(* Logix 5000 project; controller Drives_Line1 1756-L72 rev 20.13; software revision 20.04; part 6 of 21 *)
(* tags used below, declared in another part *)
   EntryCtrl : UDT_Control_Zone;
   In_Commands : UDT_Commands;
   In_Config : UDT_Config;
   In_Setpoints : UDT_Setpoints;
   LineCmd : UDT_Commands_Line;
   Out_Feedbacks : UDT_Fdbks;
   Out_Status : UDT_Status;
   TestConfig_Unwinder_1 : UDT_Config_Unwinder;
   Unwinder_1 : UDT_Unwinder;
   Unwinder_2 : UDT_Unwinder;
   zConfigFromMaster : BOOL;
(* P10_Unwinder_1, continued *)

ROUTINE R98_ToDrive   (* ladder *)
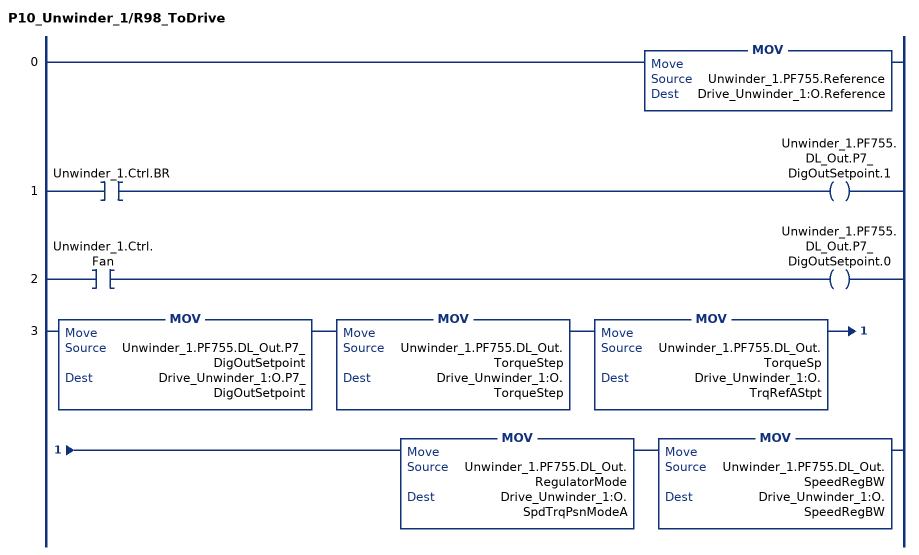
   0: MOV(Unwinder_1.PF755.Reference,Drive_Unwinder_1:O.Reference);
   1: XIC(Unwinder_1.Ctrl.BR)OTE(Unwinder_1.PF755.DL_Out.P7_DigOutSetpoint.1);
   2: XIC(Unwinder_1.Ctrl.Fan)OTE(Unwinder_1.PF755.DL_Out.P7_DigOutSetpoint.0);
   3: MOV(Unwinder_1.PF755.DL_Out.P7_DigOutSetpoint,Drive_Unwinder_1:O.P7_DigOutSetpoint)MOV(Unwinder_1.PF755.DL_Out.TorqueStep,Drive_Unwinder_1:O.TorqueStep)MOV(Unwinder_1.PF755.DL_Out.TorqueSp,Drive_Unwinder_1:O.TrqRefAStpt)MOV(Unwinder_1.PF755.DL_Out.RegulatorMode,Drive_Unwinder_1:O.SpdTrqPsnModeA)MOV(Unwinder_1.PF755.DL_Out.SpeedRegBW,Drive_Unwinder_1:O.SpeedRegBW);
END_ROUTINE

ROUTINE R999_Test   (* ladder *)
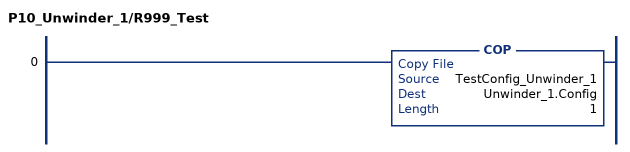
   0: COP(TestConfig_Unwinder_1,Unwinder_1.Config,1);
END_ROUTINE

ROUTINE R99_To_Master   (* ladder *)
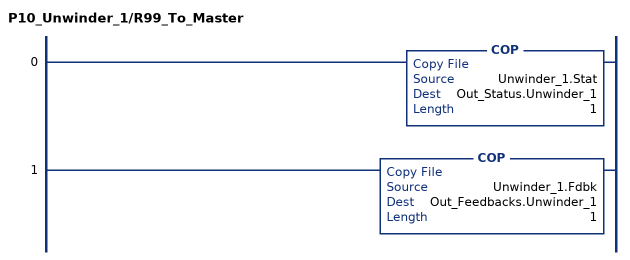
   0: COP(Unwinder_1.Stat,Out_Status.Unwinder_1,1);
   1: COP(Unwinder_1.Fdbk,Out_Feedbacks.Unwinder_1,1);
END_ROUTINE
END_PROGRAM

PROGRAM P11_Unwinder_2   (* main routine R00_Main *)
VAR
   ABS_01 : FBD_MATH_ADVANCED; {access Read Only}
   ABS_02 : FBD_MATH_ADVANCED;
   ABS_03 : FBD_MATH_ADVANCED;
   ABS_04 : FBD_MATH_ADVANCED;
   ADD_03 : FBD_MATH;
   BAND_01 : FBD_BOOLEAN_AND := (In3 := 1, In4 := 1, In5 := 1, In6 := 1, In7 := 1, In8 := 1);
   BAND_02 : FBD_BOOLEAN_AND := (In4 := 1, In5 := 1, In6 := 1, In7 := 1, In8 := 1);
   BAND_03 : FBD_BOOLEAN_AND := (In3 := 1, In4 := 1, In5 := 1, In6 := 1, In7 := 1, In8 := 1);
   BAND_04 : FBD_BOOLEAN_AND := (In3 := 1, In4 := 1, In5 := 1, In6 := 1, In7 := 1, In8 := 1);
   BAND_05 : FBD_BOOLEAN_AND := (In3 := 1, In4 := 1, In5 := 1, In6 := 1, In7 := 1, In8 := 1);
   BAND_06 : FBD_BOOLEAN_AND := (In1 := 1, In3 := 1, In4 := 1, In5 := 1, In6 := 1, In7 := 1, In8 := 1);
   BAND_07 : FBD_BOOLEAN_AND := (In3 := 1, In4 := 1, In5 := 1, In6 := 1, In7 := 1, In8 := 1);
   BAND_08 : FBD_BOOLEAN_AND := (In3 := 1, In4 := 1, In5 := 1, In6 := 1, In7 := 1, In8 := 1);
   BAND_09 : FBD_BOOLEAN_AND := (In3 := 1, In4 := 1, In5 := 1, In6 := 1, In7 := 1, In8 := 1);
   BNOT_01 : FBD_BOOLEAN_NOT := (Out := 1);
   BNOT_02 : FBD_BOOLEAN_NOT := (Out := 1);
   BNOT_04 : FBD_BOOLEAN_NOT := (Out := 1);
   BNOT_06 : FBD_BOOLEAN_NOT := (Out := 1);
   BNOT_07 : FBD_BOOLEAN_NOT := (Out := 1);
   BNOT_08 : FBD_BOOLEAN_NOT := (Out := 1);
   BOR_01 : FBD_BOOLEAN_OR := (In1 := 1, Out := 1);
   BOR_02 : FBD_BOOLEAN_OR;
   BOR_03 : FBD_BOOLEAN_OR;
   Diamtest : BOOL;
   Diamtest_mm : REAL := 725.0;
   DIV_01 : FBD_MATH := (SourceA := 2.5, SourceB := 100.0, Dest := 0.025);
   DIV_02 : FBD_MATH := (SourceB := 78.0);
   DIV_04 : FBD_MATH := (SourceB := 1440.0);
   DIV_10 : FBD_MATH := (Dest := 1770.7737);
   DIV_11 : FBD_MATH := (SourceA := 1770.7737, SourceB := 3.1415927, Dest := 563.6547);
   DIV_12 : FBD_MATH := (SourceB := 60.0);
   DIV_14 : FBD_MATH := (SourceB := 0.00494885);
   DIV_15 : FBD_MATH := (SourceA := 50.0, SourceB := 100.0, Dest := 0.5);
   EQU_01 : FBD_COMPARE := (SourceA := 1.0, SourceB := 4.0);
   FGEN_01 : FUNCTION_GENERATOR := (XY1Size := 21);
   GEQ_02 : FBD_COMPARE := (SourceB := 0.5);
   GRT_01 : FBD_COMPARE := (SourceB := 1.e-04);
   HLL_01 : HL_LIMIT := (In := 563.14075, HighLimit := 2000.0, LowLimit := 500.0, Out := 563.14075);
   HLL_07 : HL_LIMIT := (In := 6500.0, HighLimit := 15000.0, LowLimit := 1.0, Out := 6500.0);
   INTG_01 : INTEGRATOR := (Initialize := 1, IGain := 1000.02, RTSTime := 1, DeltaT := 0.05);
   INTG_02 : INTEGRATOR := (Initialize := 1, IGain := 0.016666, RTSTime := 1, DeltaT := 0.05);
   IO_State_Tmp_Unwinder_2 : INT := 16384;
   IO_State_Unwinder_2 : INT := 4;
   LES_01 : FBD_COMPARE;
   LPF_02 : FILTER_LOW_PASS := (WLag := 10.0, Order := 1, RTSTime := 1, DeltaT := 0.05); {access Read Only}
   LPF_1000 : FILTER_LOW_PASS := (WLag := 10.0, Order := 1, RTSTime := 1, DeltaT := 0.05);
   LPF_1006 : FILTER_LOW_PASS := (WLag := 10.0, Order := 1, RTSTime := 1, DeltaT := 0.05);
   MUL_01 : FBD_MATH := (SourceB := 2645.3247);
   MUL_02 : FBD_MATH := (SourceB := 0.00494885);
   MUL_03 : FBD_MATH := (SourceB := 25.0);
   MUL_04 : FBD_MATH := (SourceB := 100.0);
   MUL_05 : FBD_MATH := (SourceB := 0.5);
   MUL_06 : FBD_MATH := (SourceA := 5.0, SourceB := 0.5, Dest := 2.5);
   MUL_07 : FBD_MATH := (SourceA := 1.0065495);
   MUL_23 : FBD_MATH := (SourceA := 6500.0, SourceB := 0.5, Dest := 3250.0);
   MUL_26 : FBD_MATH := (SourceB := 2645.3247);
   NEG_01 : FBD_MATH_ADVANCED := (Source := 0.083, Dest := -0.083);
   NEG_03 : FBD_MATH_ADVANCED;
   NEG_04 : FBD_MATH_ADVANCED;
   NEG_06 : FBD_MATH_ADVANCED;
   RLIM_01 : RATE_LIMITER := (In := 563.6547, RTSTime := 1, Out := 563.14075, DeltaT := 0.05);
   RLIM_03 : RATE_LIMITER := (IncRate := 0.25, DecRate := 0.25, RTSTime := 1, DeltaT := 0.05);
   RLIM_04 : RATE_LIMITER := (IncRate := 5000.0, DecRate := 5000.0, ByPass := 1, RTSTime := 1, DeltaT := 0.05);
   SCL_01 : SCALE := (In := 562.0898, InRawMax := 5851.2163, InEUMax := 35.0, InEUMin := 25.0, Limiting := 1, Out := 25.960638);
   SCL_02 : SCALE := (InRawMax := 0.5, InEUMax := 10.0, InEUMin := 5.0, Limiting := 1, Out := 5.0);
   SCRV_02 : S_CURVE := (Initialize := 1, AbsAlgRamp := 1, AccelRate := 0.16, DecelRate := 0.16, JerkRate := 0.25, RTSTime := 1, DeltaT := 0.05);
   SEL_02 : SELECT := (In2 := 0.025);
   SEL_03 : SELECT;
   SEL_04 : SELECT;
   SEL_05 : SELECT := (In1 := 563.6547, In2 := 800.0, Out := 563.6547);
   SEL_06 : SELECT := (In1 := 563.14075, In2 := 725.0, Out := 563.14075);
   SEL_07 : SELECT := (In1 := 0.5, In2 := 0.5, Out := 0.5);
   SEL_08 : SELECT := (In1 := 563.6547, In2 := 800.0, Out := 563.6547);
   SEL_10 : SELECT;
   SEL_18 : SELECT := (In1 := 6500.0, SelectorIn := 1);
   SSUM_01 : SELECTED_SUMMER := (In1 := 0.083, Gain1 := 1.0, In2 := -0.083, Gain2 := 1.0, Gain3 := 1.0, Select3 := 1, Gain4 := 1.0, Gain5 := 1.0, Gain6 := 1.0, Gain7 := 1.0, Gain8 := 1.0);
   SSUM_02 : SELECTED_SUMMER := (Gain1 := 1.0, Select1 := 1, Gain2 := 1.0, Gain3 := 1.0, Gain4 := 1.0, Gain5 := 1.0, Gain6 := 1.0, Gain7 := 1.0, Gain8 := 1.0);
   SSUM_03 : SELECTED_SUMMER := (Gain1 := 1.0, Select1 := 1, Gain2 := 1.0, Gain3 := 1.0, Gain4 := 1.0, Gain5 := 1.0, Gain6 := 1.0, Gain7 := 1.0, Gain8 := 1.0);
   SSUM_05 : SELECTED_SUMMER := (Gain1 := 1.0, Gain2 := 1.0, Gain3 := 1.0, Gain4 := 1.0, Gain5 := 1.0, Gain6 := 1.0, Gain7 := 1.0, Gain8 := 1.0);
   SUB_08 : FBD_MATH; {access Read Only}
   TimeForBr : TIMER := (PRE := 750);
   TimeOffBr : TIMER := (PRE := 2000, ACC := 2000);
   TimeOffFan : TIMER := (PRE := 180000, ACC := 180000);
   TofReset : TIMER := (PRE := 1000, ACC := 1000);
   TonLowTension : TIMER := (PRE := 2500);
   TonNoResponse : TIMER := (PRE := 2500);
   TonRefOn : TIMER := (PRE := 500);
   TonTensionOnSp : TIMER := (PRE := 500);
   Unwind_1_DiamCalcOn : BOOL;
   Unwinder_2_JEC : REAL := 1.0; {access Read Only}
   Unwinder_2_JLossCrvSpd : REAL[21] := ([0] := -1500.0, [1] := -1350.0, [2] := -1200.0, [3] := -1050.0, [4] := -900.0, [5] := -750.0, [6] := -600.0, [7] := -450.0, [8] := -300.0, [9] := -150.0, [11] := 150.0, [12] := 300.0, [13] := 450.0, [14] := 600.0, [15] := 750.0, [16] := 900.0, [17] := 1050.0, [18] := 1200.0, [19] := 1350.0, [20] := 1500.0);
   Unwinder_2_JMaterial : REAL := 0.006549485; {access Read Only}
   Unwinder_2_LossCrvTrq_Pct : REAL[21] := ([0] := -6.0, [1] := -6.7, [2] := -6.7, [3] := -6.7, [4] := -6.7, [5] := -6.7, [6] := -6.5, [7] := -6.0, [8] := -5.0, [9] := -1.5, [11] := 2.0, [12] := 6.0, [13] := 6.8, [14] := 7.5, [15] := 7.5, [16] := 7.5, [17] := 7.5, [18] := 7.5, [19] := 7.5, [20] := 6.5);
   Unwinder_2_MatMass : REAL := 562.0898; {access Read Only}
   Unwinder_2_MatVolume : REAL := 0.15089658; {access Read Only}
   Unwinder_2_MaxMass : REAL := 5851.2163;
   Unwinder_2_MaxVolume : REAL := 1.5707964;
   Unwinder_2_PctPerN : REAL := 0.00494885; {access Read Only}
   Unwinder_2_RatedTrq : REAL := 72.94375; {access Read Only}
   Unwinder_2_RPMPerMPS : REAL := 2645.3247;
   Unwinder_2_SpdMps_Flt : REAL;
   Unwinder_2_SpdRpm_Flt : REAL;
   zUnwind_2_MaxRate : REAL := 0.25;
   zUnwind_2_TenRefRate : REAL := 5000.0;
   zUnwind_2_TenSpStall : REAL := 50.0;
   zUnwind_2_TrqTrimLimMax_Pct : REAL := 10.0;
   zUnwind_2_TrqTrimLimMin_Pct : REAL := 5.0;
   zUnwinder_2_JGainQ1Q2 : REAL := 0.5;
   zUnwinder_2_JGainQ3Q4 : REAL := 0.5;
   zUnwinder_2_SpdReg_BWMax : REAL := 35.0;
   zUnwinder_2_SpdReg_BWmin : REAL := 25.0;
   zUnwinder_2_Stall_Spd : REAL := 5.0;
   zUnwinder_2_Tens_Offs : REAL := 100.0;
END_VAR

ROUTINE R00_Main   (* ladder *)
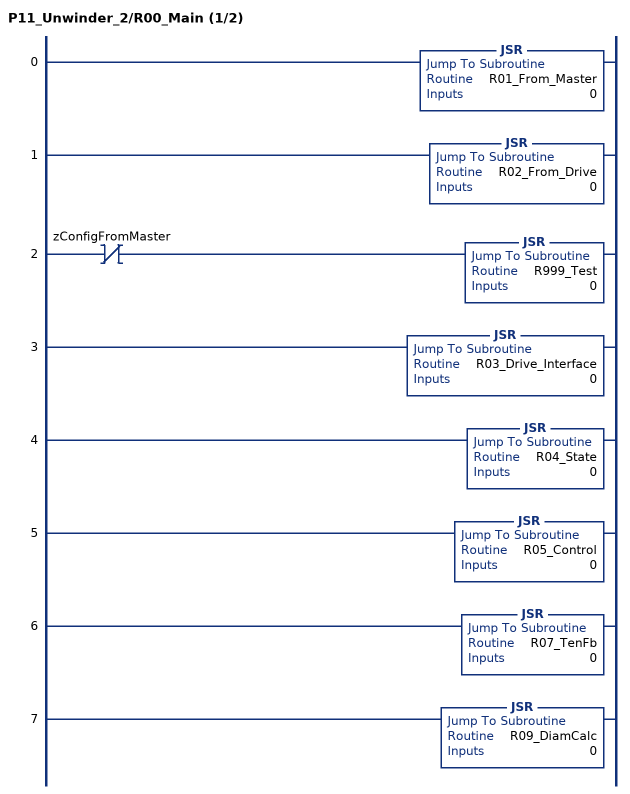
   0: JSR(R01_From_Master,0);
   1: JSR(R02_From_Drive,0);
   2: XIO(zConfigFromMaster)JSR(R999_Test,0);
   3: JSR(R03_Drive_Interface,0);
   4: JSR(R04_State,0);
   5: JSR(R05_Control,0);
   6: JSR(R07_TenFb,0);
   7: JSR(R09_DiamCalc,0);
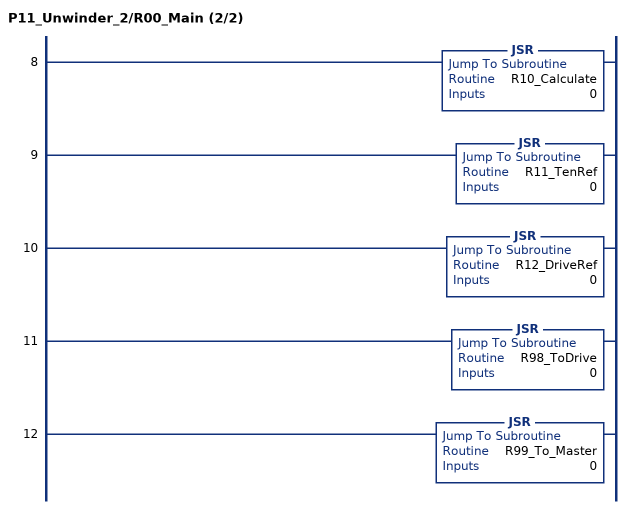
   8: JSR(R10_Calculate,0);
   9: JSR(R11_TenRef,0);
   10: JSR(R12_DriveRef,0);
   11: JSR(R98_ToDrive,0);
   12: JSR(R99_To_Master,0);
END_ROUTINE

ROUTINE R01_From_Master   (* ladder *)
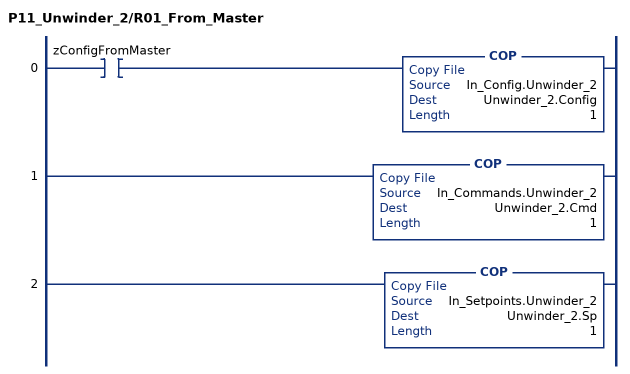
   0: XIC(zConfigFromMaster)COP(In_Config.Unwinder_2,Unwinder_2.Config,1);
   1: COP(In_Commands.Unwinder_2,Unwinder_2.Cmd,1);
   2: COP(In_Setpoints.Unwinder_2,Unwinder_2.Sp,1);
END_ROUTINE

ROUTINE R02_From_Drive   (* ladder *)
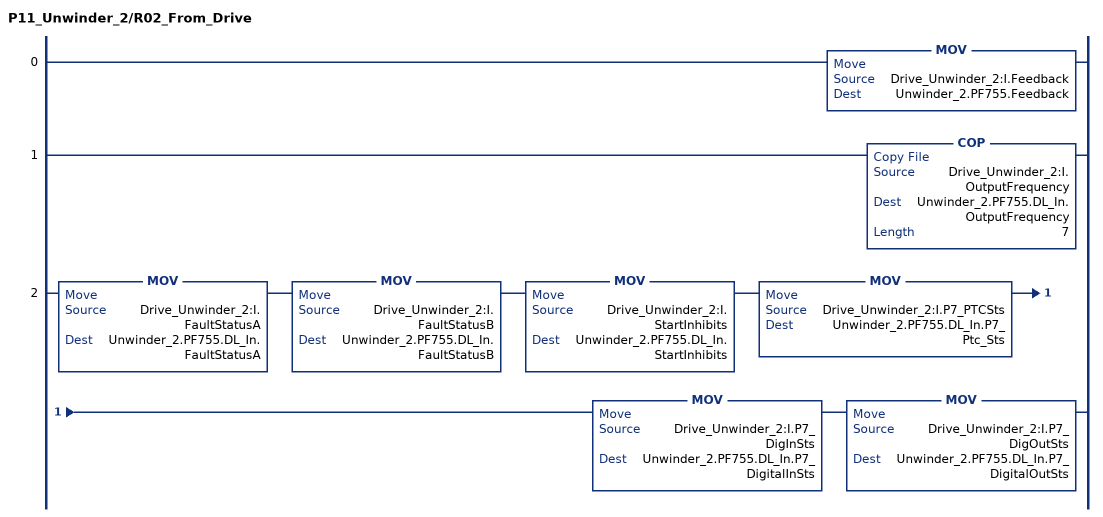
   0: MOV(Drive_Unwinder_2:I.Feedback,Unwinder_2.PF755.Feedback);
   1: COP(Drive_Unwinder_2:I.OutputFrequency,Unwinder_2.PF755.DL_In.OutputFrequency,7);
   2: MOV(Drive_Unwinder_2:I.FaultStatusA,Unwinder_2.PF755.DL_In.FaultStatusA)MOV(Drive_Unwinder_2:I.FaultStatusB,Unwinder_2.PF755.DL_In.FaultStatusB)MOV(Drive_Unwinder_2:I.StartInhibits,Unwinder_2.PF755.DL_In.StartInhibits)MOV(Drive_Unwinder_2:I.P7_PTCSts,Unwinder_2.PF755.DL_In.P7_Ptc_Sts)MOV(Drive_Unwinder_2:I.P7_DigInSts,Unwinder_2.PF755.DL_In.P7_DigitalInSts)MOV(Drive_Unwinder_2:I.P7_DigOutSts,Unwinder_2.PF755.DL_In.P7_DigitalOutSts);
END_ROUTINE

ROUTINE R03_Drive_Interface   (* ladder *)
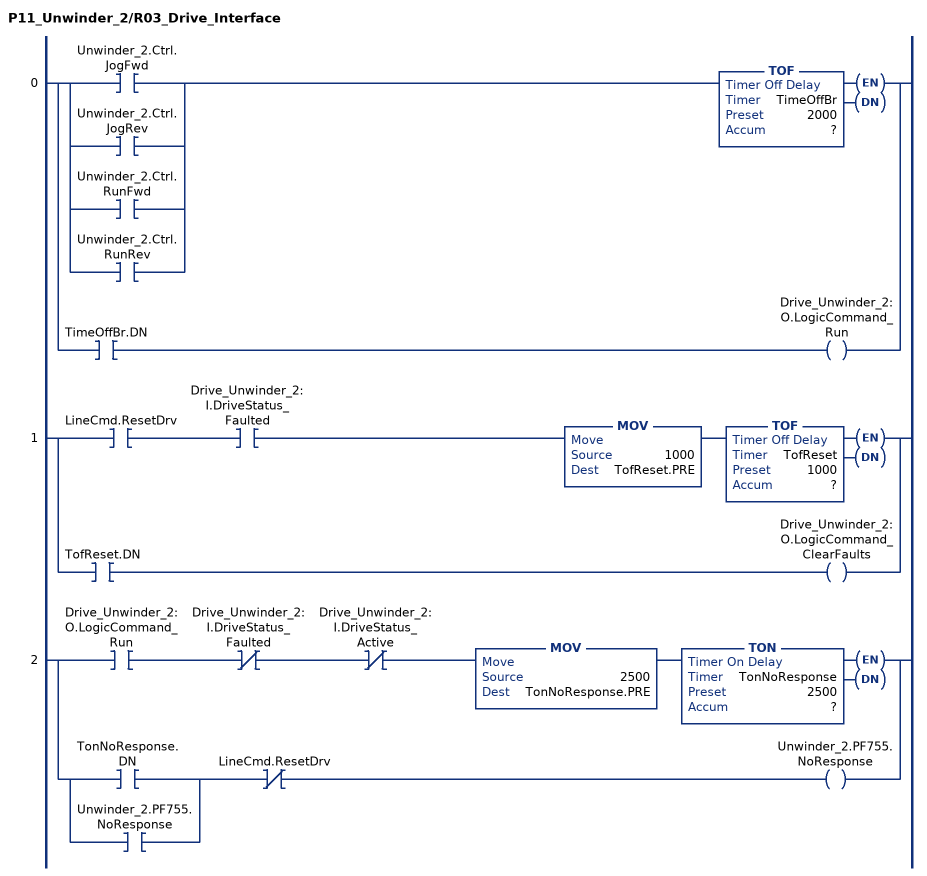
   0: [[XIC(Unwinder_2.Ctrl.JogFwd) ,XIC(Unwinder_2.Ctrl.JogRev) ,XIC(Unwinder_2.Ctrl.RunFwd) ,XIC(Unwinder_2.Ctrl.RunRev) ] TOF(TimeOffBr,?,?) ,XIC(TimeOffBr.DN) OTE(Drive_Unwinder_2:O.LogicCommand_Run) ];
   1: [XIC(LineCmd.ResetDrv) XIC(Drive_Unwinder_2:I.DriveStatus_Faulted) MOV(1000,TofReset.PRE) TOF(TofReset,?,?) ,XIC(TofReset.DN) OTE(Drive_Unwinder_2:O.LogicCommand_ClearFaults) ];
   2: [XIC(Drive_Unwinder_2:O.LogicCommand_Run) XIO(Drive_Unwinder_2:I.DriveStatus_Faulted) XIO(Drive_Unwinder_2:I.DriveStatus_Active) MOV(2500,TonNoResponse.PRE) TON(TonNoResponse,?,?) ,[XIC(TonNoResponse.DN) ,XIC(Unwinder_2.PF755.NoResponse) ] XIO(LineCmd.ResetDrv) OTE(Unwinder_2.PF755.NoResponse) ];
END_ROUTINE

ROUTINE R04_State   (* ladder *)
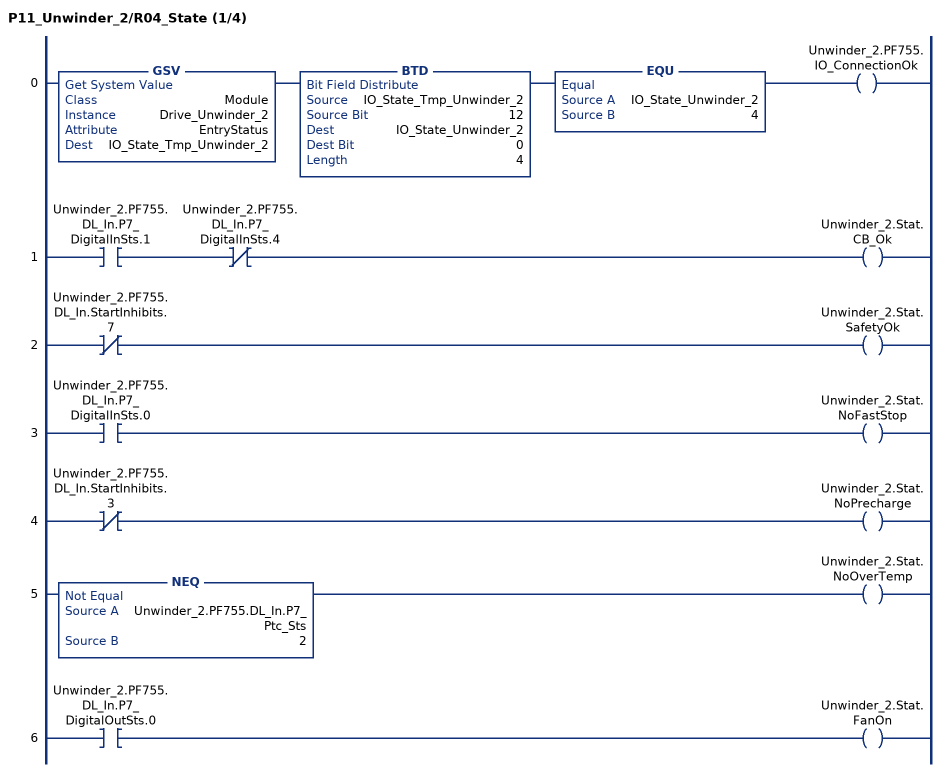
   0: GSV(Module,Drive_Unwinder_2,EntryStatus,IO_State_Tmp_Unwinder_2)BTD(IO_State_Tmp_Unwinder_2,12,IO_State_Unwinder_2,0,4)EQU(IO_State_Unwinder_2,4)OTE(Unwinder_2.PF755.IO_ConnectionOk);
   1: XIC(Unwinder_2.PF755.DL_In.P7_DigitalInSts.1)XIO(Unwinder_2.PF755.DL_In.P7_DigitalInSts.4)OTE(Unwinder_2.Stat.CB_Ok);
   2: XIO(Unwinder_2.PF755.DL_In.StartInhibits.7)OTE(Unwinder_2.Stat.SafetyOk);
   3: XIC(Unwinder_2.PF755.DL_In.P7_DigitalInSts.0)OTE(Unwinder_2.Stat.NoFastStop);
   4: XIO(Unwinder_2.PF755.DL_In.StartInhibits.3)OTE(Unwinder_2.Stat.NoPrecharge);
   5: NEQ(Unwinder_2.PF755.DL_In.P7_Ptc_Sts,2)OTE(Unwinder_2.Stat.NoOverTemp);
   6: XIC(Unwinder_2.PF755.DL_In.P7_DigitalOutSts.0)OTE(Unwinder_2.Stat.FanOn);
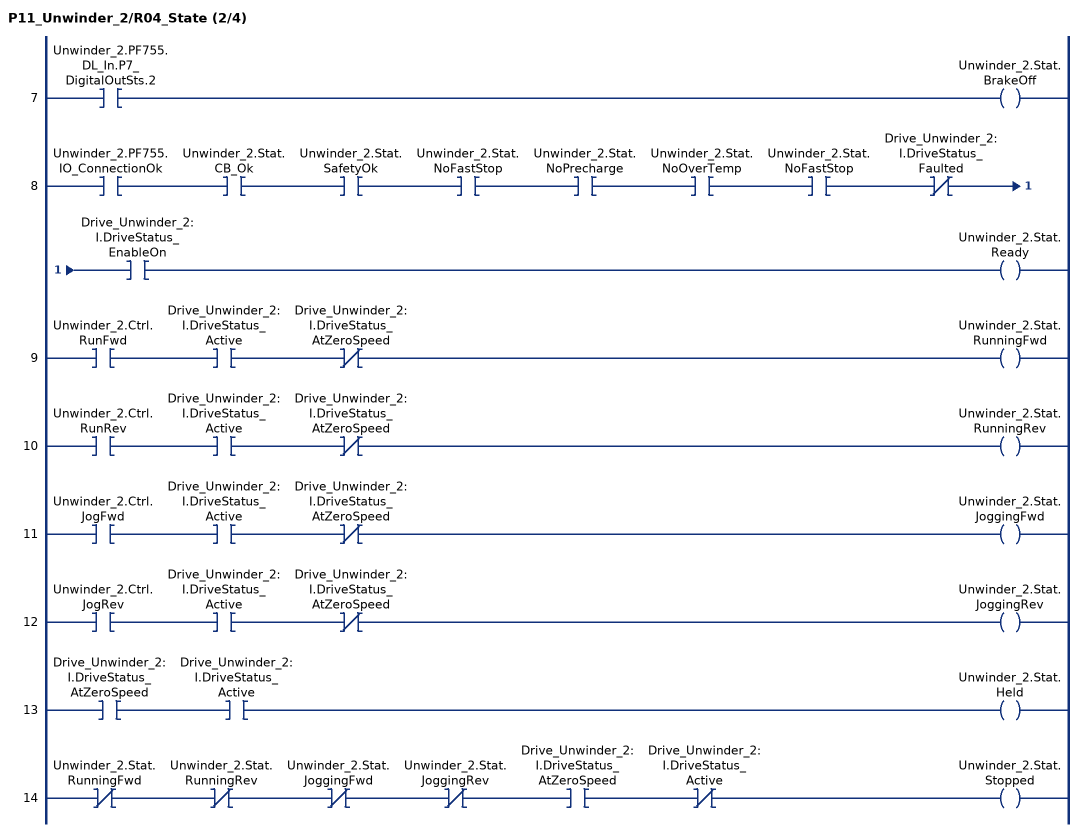
   7: XIC(Unwinder_2.PF755.DL_In.P7_DigitalOutSts.2)OTE(Unwinder_2.Stat.BrakeOff);
   8: XIC(Unwinder_2.PF755.IO_ConnectionOk)XIC(Unwinder_2.Stat.CB_Ok)XIC(Unwinder_2.Stat.SafetyOk)XIC(Unwinder_2.Stat.NoFastStop)XIC(Unwinder_2.Stat.NoPrecharge)XIC(Unwinder_2.Stat.NoOverTemp)XIC(Unwinder_2.Stat.NoFastStop)XIO(Drive_Unwinder_2:I.DriveStatus_Faulted)XIC(Drive_Unwinder_2:I.DriveStatus_EnableOn)OTE(Unwinder_2.Stat.Ready);
   9: XIC(Unwinder_2.Ctrl.RunFwd)XIC(Drive_Unwinder_2:I.DriveStatus_Active)XIO(Drive_Unwinder_2:I.DriveStatus_AtZeroSpeed)OTE(Unwinder_2.Stat.RunningFwd);
   10: XIC(Unwinder_2.Ctrl.RunRev)XIC(Drive_Unwinder_2:I.DriveStatus_Active)XIO(Drive_Unwinder_2:I.DriveStatus_AtZeroSpeed)OTE(Unwinder_2.Stat.RunningRev);
   11: XIC(Unwinder_2.Ctrl.JogFwd)XIC(Drive_Unwinder_2:I.DriveStatus_Active)XIO(Drive_Unwinder_2:I.DriveStatus_AtZeroSpeed)OTE(Unwinder_2.Stat.JoggingFwd);
   12: XIC(Unwinder_2.Ctrl.JogRev)XIC(Drive_Unwinder_2:I.DriveStatus_Active)XIO(Drive_Unwinder_2:I.DriveStatus_AtZeroSpeed)OTE(Unwinder_2.Stat.JoggingRev);
   13: XIC(Drive_Unwinder_2:I.DriveStatus_AtZeroSpeed)XIC(Drive_Unwinder_2:I.DriveStatus_Active)OTE(Unwinder_2.Stat.Held);
   14: XIO(Unwinder_2.Stat.RunningFwd)XIO(Unwinder_2.Stat.RunningRev)XIO(Unwinder_2.Stat.JoggingFwd)XIO(Unwinder_2.Stat.JoggingRev)XIC(Drive_Unwinder_2:I.DriveStatus_AtZeroSpeed)XIO(Drive_Unwinder_2:I.DriveStatus_Active)OTE(Unwinder_2.Stat.Stopped);
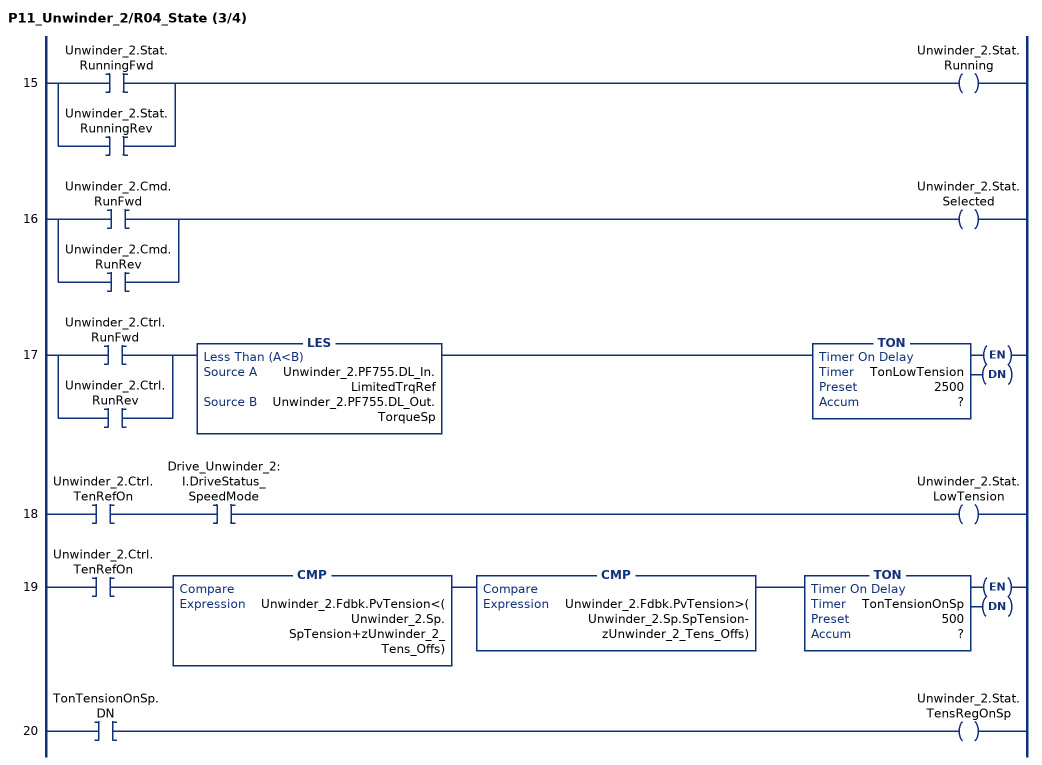
   15: [XIC(Unwinder_2.Stat.RunningFwd) ,XIC(Unwinder_2.Stat.RunningRev) ]OTE(Unwinder_2.Stat.Running);
   16: [XIC(Unwinder_2.Cmd.RunFwd) ,XIC(Unwinder_2.Cmd.RunRev) ]OTE(Unwinder_2.Stat.Selected);
   17: [XIC(Unwinder_2.Ctrl.RunFwd) ,XIC(Unwinder_2.Ctrl.RunRev) ]LES(Unwinder_2.PF755.DL_In.LimitedTrqRef,Unwinder_2.PF755.DL_Out.TorqueSp)TON(TonLowTension,?,?);
   18: XIC(Unwinder_2.Ctrl.TenRefOn)XIC(Drive_Unwinder_2:I.DriveStatus_SpeedMode)OTE(Unwinder_2.Stat.LowTension);
   19: XIC(Unwinder_2.Ctrl.TenRefOn)CMP(Unwinder_2.Fdbk.PvTension<(Unwinder_2.Sp.SpTension+zUnwinder_2_Tens_Offs))CMP(Unwinder_2.Fdbk.PvTension>(Unwinder_2.Sp.SpTension-zUnwinder_2_Tens_Offs))TON(TonTensionOnSp,?,?);
   20: XIC(TonTensionOnSp.DN)OTE(Unwinder_2.Stat.TensRegOnSp);
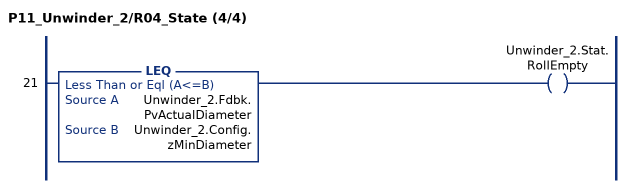
   21: LEQ(Unwinder_2.Fdbk.PvActualDiameter,Unwinder_2.Config.zMinDiameter)OTE(Unwinder_2.Stat.RollEmpty);
END_ROUTINE

ROUTINE R05_Control   (* ladder *)
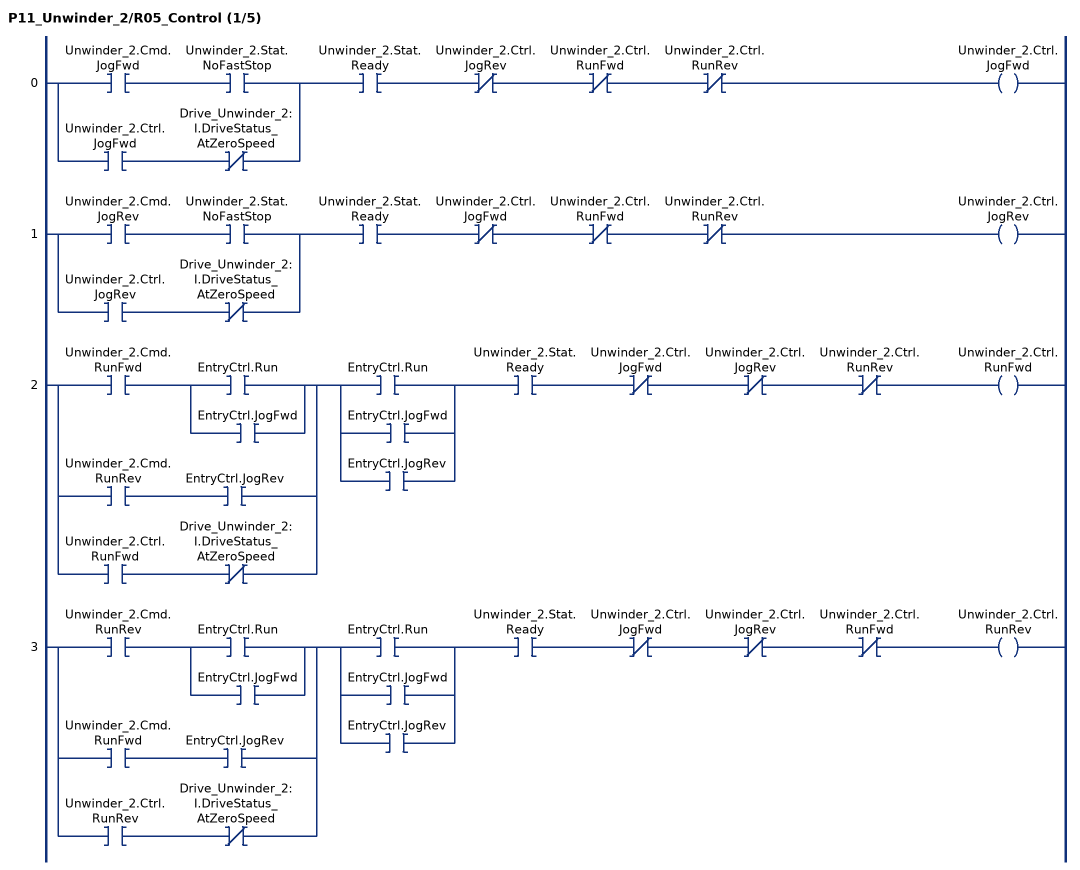
   0: [XIC(Unwinder_2.Cmd.JogFwd) XIC(Unwinder_2.Stat.NoFastStop) ,XIC(Unwinder_2.Ctrl.JogFwd) XIO(Drive_Unwinder_2:I.DriveStatus_AtZeroSpeed) ]XIC(Unwinder_2.Stat.Ready)XIO(Unwinder_2.Ctrl.JogRev)XIO(Unwinder_2.Ctrl.RunFwd)XIO(Unwinder_2.Ctrl.RunRev)OTE(Unwinder_2.Ctrl.JogFwd);
   1: [XIC(Unwinder_2.Cmd.JogRev) XIC(Unwinder_2.Stat.NoFastStop) ,XIC(Unwinder_2.Ctrl.JogRev) XIO(Drive_Unwinder_2:I.DriveStatus_AtZeroSpeed) ]XIC(Unwinder_2.Stat.Ready)XIO(Unwinder_2.Ctrl.JogFwd)XIO(Unwinder_2.Ctrl.RunFwd)XIO(Unwinder_2.Ctrl.RunRev)OTE(Unwinder_2.Ctrl.JogRev);
   2: [XIC(Unwinder_2.Cmd.RunFwd) [XIC(EntryCtrl.Run) ,XIC(EntryCtrl.JogFwd) ] ,XIC(Unwinder_2.Cmd.RunRev) XIC(EntryCtrl.JogRev) ,XIC(Unwinder_2.Ctrl.RunFwd) XIO(Drive_Unwinder_2:I.DriveStatus_AtZeroSpeed) ][XIC(EntryCtrl.Run) ,XIC(EntryCtrl.JogFwd) ,XIC(EntryCtrl.JogRev) ]XIC(Unwinder_2.Stat.Ready)XIO(Unwinder_2.Ctrl.JogFwd)XIO(Unwinder_2.Ctrl.JogRev)XIO(Unwinder_2.Ctrl.RunRev)OTE(Unwinder_2.Ctrl.RunFwd);
   3: [XIC(Unwinder_2.Cmd.RunRev) [XIC(EntryCtrl.Run) ,XIC(EntryCtrl.JogFwd) ] ,XIC(Unwinder_2.Cmd.RunFwd) XIC(EntryCtrl.JogRev) ,XIC(Unwinder_2.Ctrl.RunRev) XIO(Drive_Unwinder_2:I.DriveStatus_AtZeroSpeed) ][XIC(EntryCtrl.Run) ,XIC(EntryCtrl.JogFwd) ,XIC(EntryCtrl.JogRev) ]XIC(Unwinder_2.Stat.Ready)XIO(Unwinder_2.Ctrl.JogFwd)XIO(Unwinder_2.Ctrl.JogRev)XIO(Unwinder_2.Ctrl.RunFwd)OTE(Unwinder_2.Ctrl.RunRev);
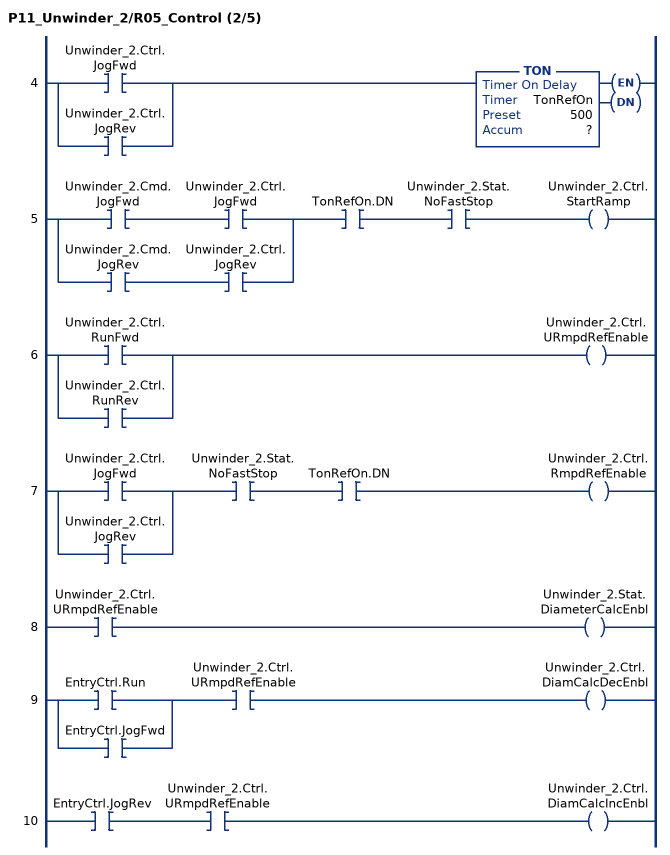
   4: [XIC(Unwinder_2.Ctrl.JogFwd) ,XIC(Unwinder_2.Ctrl.JogRev) ]TON(TonRefOn,?,?);
   5: [XIC(Unwinder_2.Cmd.JogFwd) XIC(Unwinder_2.Ctrl.JogFwd) ,XIC(Unwinder_2.Cmd.JogRev) XIC(Unwinder_2.Ctrl.JogRev) ]XIC(TonRefOn.DN)XIC(Unwinder_2.Stat.NoFastStop)OTE(Unwinder_2.Ctrl.StartRamp);
   6: [XIC(Unwinder_2.Ctrl.RunFwd) ,XIC(Unwinder_2.Ctrl.RunRev) ]OTE(Unwinder_2.Ctrl.URmpdRefEnable);
   7: [XIC(Unwinder_2.Ctrl.JogFwd) ,XIC(Unwinder_2.Ctrl.JogRev) ]XIC(Unwinder_2.Stat.NoFastStop)XIC(TonRefOn.DN)OTE(Unwinder_2.Ctrl.RmpdRefEnable);
   8: XIC(Unwinder_2.Ctrl.URmpdRefEnable)OTE(Unwinder_2.Stat.DiameterCalcEnbl);
   9: [XIC(EntryCtrl.Run) ,XIC(EntryCtrl.JogFwd) ]XIC(Unwinder_2.Ctrl.URmpdRefEnable)OTE(Unwinder_2.Ctrl.DiamCalcDecEnbl);
   10: XIC(EntryCtrl.JogRev)XIC(Unwinder_2.Ctrl.URmpdRefEnable)OTE(Unwinder_2.Ctrl.DiamCalcIncEnbl);
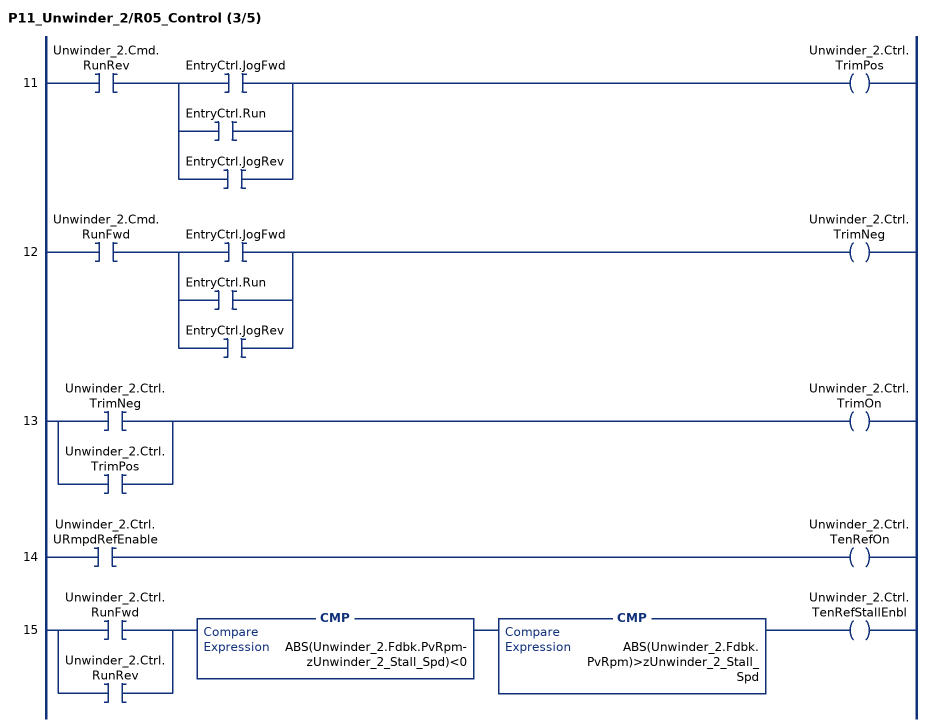
   11: XIC(Unwinder_2.Cmd.RunRev)[XIC(EntryCtrl.JogFwd) ,XIC(EntryCtrl.Run) ,XIC(EntryCtrl.JogRev) ]OTE(Unwinder_2.Ctrl.TrimPos);
   12: XIC(Unwinder_2.Cmd.RunFwd)[XIC(EntryCtrl.JogFwd) ,XIC(EntryCtrl.Run) ,XIC(EntryCtrl.JogRev) ]OTE(Unwinder_2.Ctrl.TrimNeg);
   13: [XIC(Unwinder_2.Ctrl.TrimNeg) ,XIC(Unwinder_2.Ctrl.TrimPos) ]OTE(Unwinder_2.Ctrl.TrimOn);
   14: XIC(Unwinder_2.Ctrl.URmpdRefEnable)OTE(Unwinder_2.Ctrl.TenRefOn);
   15: [XIC(Unwinder_2.Ctrl.RunFwd) ,XIC(Unwinder_2.Ctrl.RunRev) ]CMP(ABS(Unwinder_2.Fdbk.PvRpm-zUnwinder_2_Stall_Spd)<0)CMP(ABS(Unwinder_2.Fdbk.PvRpm)>zUnwinder_2_Stall_Spd)OTE(Unwinder_2.Ctrl.TenRefStallEnbl);
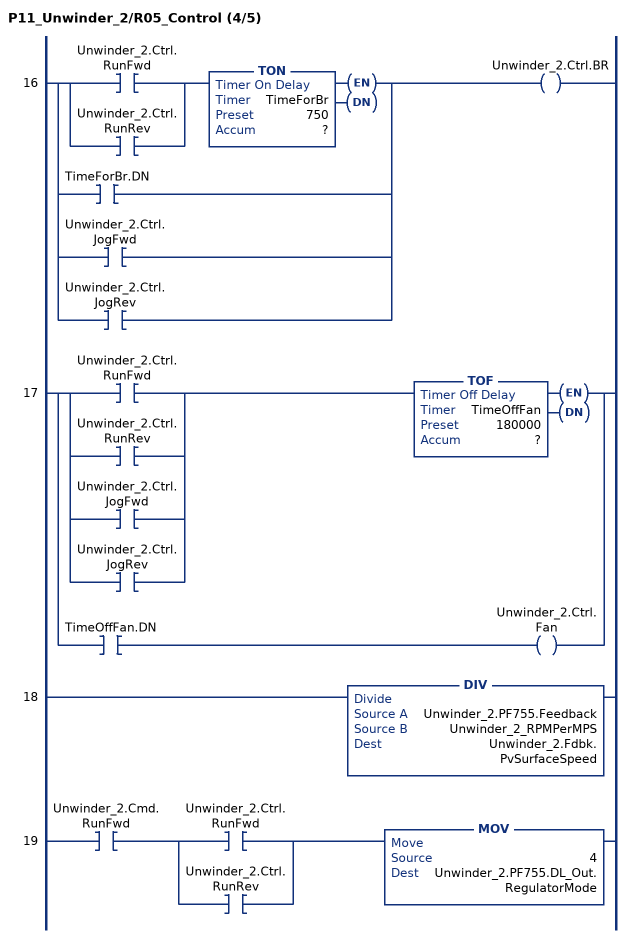
   16: [[XIC(Unwinder_2.Ctrl.RunFwd) ,XIC(Unwinder_2.Ctrl.RunRev) ] TON(TimeForBr,?,?) ,XIC(TimeForBr.DN) ,XIC(Unwinder_2.Ctrl.JogFwd) ,XIC(Unwinder_2.Ctrl.JogRev) ]OTE(Unwinder_2.Ctrl.BR);
   17: [[XIC(Unwinder_2.Ctrl.RunFwd) ,XIC(Unwinder_2.Ctrl.RunRev) ,XIC(Unwinder_2.Ctrl.JogFwd) ,XIC(Unwinder_2.Ctrl.JogRev) ] TOF(TimeOffFan,?,?) ,XIC(TimeOffFan.DN) OTE(Unwinder_2.Ctrl.Fan) ];
   18: DIV(Unwinder_2.PF755.Feedback,Unwinder_2_RPMPerMPS,Unwinder_2.Fdbk.PvSurfaceSpeed);
   19: XIC(Unwinder_2.Cmd.RunFwd)[XIC(Unwinder_2.Ctrl.RunFwd) ,XIC(Unwinder_2.Ctrl.RunRev) ]MOV(4,Unwinder_2.PF755.DL_Out.RegulatorMode);
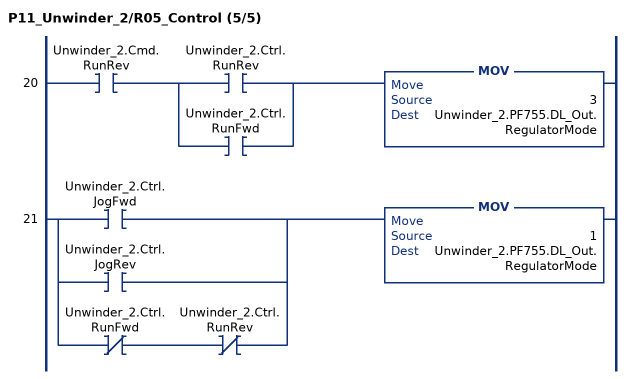
   20: XIC(Unwinder_2.Cmd.RunRev)[XIC(Unwinder_2.Ctrl.RunRev) ,XIC(Unwinder_2.Ctrl.RunFwd) ]MOV(3,Unwinder_2.PF755.DL_Out.RegulatorMode);
   21: [XIC(Unwinder_2.Ctrl.JogFwd) ,XIC(Unwinder_2.Ctrl.JogRev) ,XIO(Unwinder_2.Ctrl.RunFwd) XIO(Unwinder_2.Ctrl.RunRev) ]MOV(1,Unwinder_2.PF755.DL_Out.RegulatorMode);
END_ROUTINE

ROUTINE R07_TenFb   (* function block diagram *)
   SHEET 1   // Torque Feedback
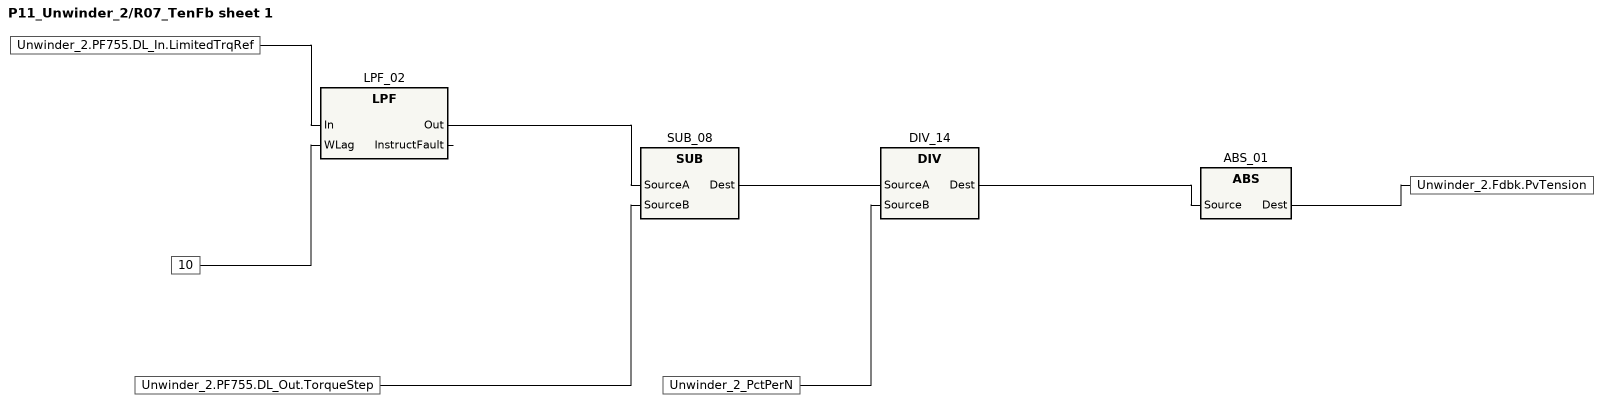
   LPF_02 : LPF(In := Unwinder_2.PF755.DL_In.LimitedTrqRef, WLag := 10);   // unwired pins: InstructFault
   SUB_08 : SUB(SourceA := LPF_02.Out, SourceB := Unwinder_2.PF755.DL_Out.TorqueStep);
   DIV_14 : DIV(SourceA := SUB_08.Dest, SourceB := Unwinder_2_PctPerN);
   ABS_01 : ABS(Source := DIV_14.Dest);
   Unwinder_2.Fdbk.PvTension := ABS_01.Dest;
   SHEET 2   // Speed Feedback
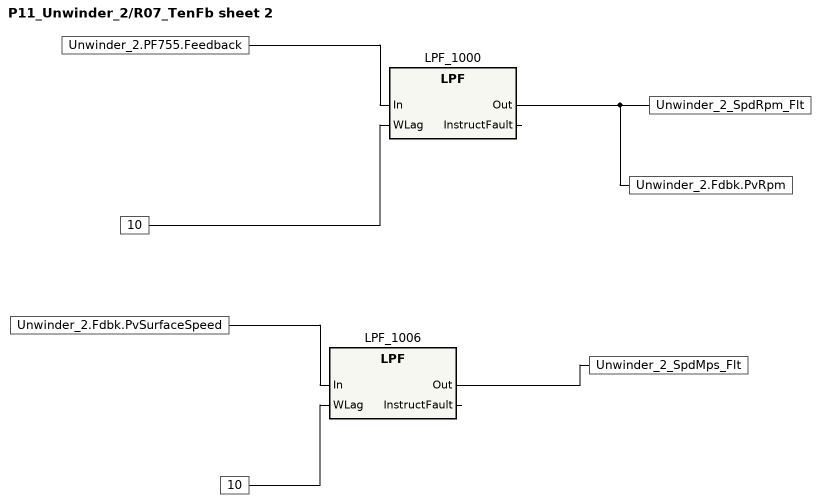
   LPF_1006 : LPF(In := Unwinder_2.Fdbk.PvSurfaceSpeed, WLag := 10);   // unwired pins: InstructFault
   LPF_1000 : LPF(In := Unwinder_2.PF755.Feedback, WLag := 10);   // unwired pins: InstructFault
   Unwinder_2_SpdMps_Flt := LPF_1006.Out;
   Unwinder_2.Fdbk.PvRpm := LPF_1000.Out;
   Unwinder_2_SpdRpm_Flt := LPF_1000.Out;
END_ROUTINE
